IF Reporter = 0 THEN
	RETURN;
END_IF

IF _ReporterCount >= TestHarnessParameter.ReporterCapacity THEN
	THIS^.RaiseFrameworkError('the run cannot hold another reporter');
	RETURN;
END_IF

_Reporters[TO_DINT(_ReporterCount)] := Reporter;
_ReporterCount := _ReporterCount + 1;

_Fanout.Attach(Reporter);

// Suites added before this reporter was.
FOR i := 0 TO TO_DINT(_Count) - 1 DO
	THIS^.PushReporter(_Suites[i], Reporter);
END_FOR

AddReporter := TRUE;
END_METHOD

PROPERTY ReporterCount : UDINT
GET
ReporterCount := _Fanout.Count;
END_GET
END_PROPERTY

METHOD SetLabel
VAR_INPUT
	Label : T_MaxString;
END_VAR
_Label := Label;
_Tally.SetLabel(Label);
END_METHOD

// Drive the run. One suite at a time, in the order they were added.
//
// Returns TRUE once every suite has reached a terminal state.
METHOD Run : BOOL
VAR_INPUT
	Enable : BOOL;
END_VAR

VAR
	Index : DINT;
END_VAR
_Fanout.CyclicLogic();

Run := _Tally.IsComplete;

IF NOT Enable THEN
	RETURN;
END_IF

IF _IsOpen THEN
	_IsOpen := FALSE;
	THIS^.BeginTally();

	IF _Label = '' THEN
		THIS^.RaiseFrameworkError('the run was started with no label');
	END_IF

	// Once, before anything else in the run. A sink that builds something opens it
	// here rather than guessing from the first result to arrive.
	_Fanout.RunStarted(Label := _Label, TargetInfo := _TargetInfo);
END_IF

IF _Tally.IsComplete THEN
	RETURN;
END_IF

IF _Index >= TO_DINT(_Count) THEN
	THIS^.Finish();
	Run := _Tally.IsComplete;
	RETURN;
END_IF

Index := _Index;

// Serial by construction. Only one suite is ever enabled, which is what makes two
// suites touching the same axis unable to overlap.
IF _Suites[Index].Run(Enable := TRUE) THEN
	// Counts TESTS, not suites, so the figures mean the same thing at every level
	// of a nest.
	_Tally.Absorb(_Suites[Index]);
	THIS^.NextSuite();
ELSE
	THIS^.CheckWatchdog(Index);
END_IF

Run := _Tally.IsComplete;
END_METHOD

// Nothing to run. The run reports complete rather than waiting, so anything
// aggregating it is not held open.
METHOD Skip
IF NOT _IsOpen THEN
	RETURN;
END_IF

_IsOpen := FALSE;
_Tally.Begin(0);
_Index	:= TO_DINT(_Count);
THIS^.Finish();
END_METHOD

// Add a suite to the run. Order of addition is order of execution.
//
// That ordering is what gives coarse exclusion for free: two integration suites
// touching the same axis cannot overlap, because only one is ever enabled.
METHOD AddSuite : BOOL
VAR_INPUT
	Suite : I_TestSuite;
END_VAR

VAR
	Index : DINT;
	i	  : DINT;
END_VAR
AddSuite := FALSE;

IF Suite = 0 THEN
	THIS^.RaiseFrameworkError('a null suite was offered');
	RETURN;
END_IF

IF NOT _IsOpen THEN
	THIS^.RaiseFrameworkError('suites cannot be added once the run has started');
	RETURN;
END_IF

IF _Count >= Capacity THEN
	THIS^.RaiseFrameworkError('the run is full - raise its capacity argument');
	RETURN;
END_IF

Index		 := TO_DINT(_Count);
_Suites[Index] := Suite;
_Count		 := _Count + 1;

// Reporters already attached reach this suite too, so the composition root
// attaches once - to the run - whatever order it does things in.
FOR i := 0 TO TO_DINT(_ReporterCount) - 1 DO
	THIS^.PushReporter(Suite, _Reporters[i]);
END_FOR

AddSuite := TRUE;
END_METHOD

// Suites added. Assert it in CI: a suite that silently stops being added takes
// its tests with it, and the totals simply come out smaller.
PROPERTY SuiteCount : UDINT
GET
SuiteCount := _Count;
END_GET
END_PROPERTY

PROPERTY ErrorCount : UDINT
GET
ErrorCount := _Tally.ErrorCount;
END_GET
END_PROPERTY

PROPERTY FailedCount : UDINT
GET
FailedCount := _Tally.FailedCount;
END_GET
END_PROPERTY

PROPERTY IsComplete : BOOL
GET
IsComplete := _Tally.IsComplete;
END_GET
END_PROPERTY

PROPERTY Outcome : E_RunOutcome
GET
Outcome := _Tally.Outcome;
END_GET
END_PROPERTY

PROPERTY PassedCount : UDINT
GET
PassedCount := _Tally.PassedCount;
END_GET
END_PROPERTY

PROPERTY SkippedCount : UDINT
GET
SkippedCount := _Tally.SkippedCount;
END_GET
END_PROPERTY

PROPERTY TestCount : UDINT
GET
TestCount := _Tally.TestCount;
END_GET
END_PROPERTY

PROPERTY TotalDuration : LREAL
GET
TotalDuration := _Tally.TotalDuration;
END_GET
END_PROPERTY

// Start the aggregate, and re-apply anything raised before it existed.
//
// A framework error raised while the run was still OPEN - a refused suite, a
// refused reporter - has no tally to record itself into. It is counted in
// _PendingErrors and re-applied here, or a run that could not be composed
// properly reports green with its missing tests simply absent from the totals.
//
// ORDER MATTERS: Begin clears ErrorCount, so the drain must follow it. Both entry
// points into a run go through this method for that reason.
//
// _PendingErrors is NOT cleared. A suite that failed to be added is still missing
// on a re-run, so the error is re-applied every time the aggregate restarts.
METHOD BeginTally
VAR
	i : DINT;
END_VAR
_Tally.Begin(0);

FOR i := 1 TO TO_DINT(_PendingErrors) DO
	_Tally.RecordFrameworkError();
END_FOR
END_METHOD

// Has the active suite stopped making progress?
//
// PROGRESS, not duration. The measure is how many tests the suite has brought to
// a verdict - passed, failed, errored or skipped. A slow suite still moves that
// number; a stalled one does not, and counting scans since it STARTED would fire
// on the slow rather than the stuck.
//
// A suite cannot see this about itself: it is the thing that has stopped. The run
// owns the sequence, so it is the only object positioned to notice.
METHOD CheckWatchdog
VAR_INPUT
	Index : DINT;
END_VAR

VAR
	Progress : UDINT;
	Suite	 : I_TestSuite;
END_VAR
IF _WatchdogCycles = 0 THEN
	RETURN;
END_IF

Suite := _Suites[Index];

IF Suite = 0 THEN
	RETURN;
END_IF

// Every verdict the suite has reached so far.
Progress := Suite.PassedCount + Suite.FailedCount
		  + Suite.ErrorCount + Suite.SkippedCount;

IF Progress <> _LastProgress THEN
	_LastProgress := Progress;
	_StallCycles  := 0;
	RETURN;
END_IF

_StallCycles := _StallCycles + 1;

IF _StallCycles < _WatchdogCycles THEN
	RETURN;
END_IF

// Stalled. Named, counted, and left behind.
_StalledSuites := _StalledSuites + 1;
THIS^.RaiseFrameworkError(CONCAT(CONCAT(
	'suite stalled and was abandoned: ', Suite.Label),
	CONCAT(', no verdict for ', UDINT_TO_STRING(_WatchdogCycles))));

// One call with Enable FALSE, so the suite can put its own state back. Its return
// is ignored: a suite that has stopped will not answer this either, and waiting
// for it would reproduce the stall the watchdog exists to break.
Suite.Run(Enable := FALSE);

// Whatever it did manage still counts.
_Tally.Absorb(Suite);

THIS^.NextSuite();
END_METHOD

// Terminal. Settles the aggregate and raises RunFinished - ONCE, whatever the
// topology.
//
// THIS IS WHY THIS OBJECT EXISTS. A suite cannot raise it: a suite is not a run,
// and asking one to announce the end of something above itself is what forced a
// "am I being sequenced" flag in an earlier design. Here a single suite is
// composed with one TestRun and a sequencer IS one, so exactly one object is ever
// in a position to say the run is over.
METHOD Finish
IF _Tally.IsComplete THEN
	RETURN;
END_IF

_Tally.Finish();
_Fanout.RunFinished(Status := THIS^, TargetInfo := _TargetInfo);
END_METHOD

// Move to the next suite and reset the watchdog with it. One place, so the reset
// cannot be forgotten on one of the paths that advances.
METHOD NextSuite
_Index		  := _Index + 1;
_StallCycles  := 0;
_LastProgress := 0;
END_METHOD

// Hand a reporter to a suite through its configuration face.
//
// A suite is held as I_TestSuite - the driving surface - which deliberately does
// not carry AddReporter. The configuration face is reached with __QUERYINTERFACE,
// the same way every optional face in this library is.
METHOD PushReporter
VAR_INPUT
	Suite	 : I_TestSuite;
	Reporter : I_TestReporter;
END_VAR

VAR
	ConfigFace : I_TestConfiguration;
END_VAR
IF Suite = 0 THEN
	RETURN;
END_IF

IF __QUERYINTERFACE(Suite, ConfigFace) THEN
	ConfigFace.AddReporter(Reporter);
END_IF
END_METHOD

// One place run-level framework errors are named.
METHOD RaiseFrameworkError
VAR_INPUT
	Message : T_MaxString;
END_VAR
IF _IsOpen THEN
	// Before the tally exists. Held, and re-applied by BeginTally when the run
	// starts - without that, a run that could not be composed properly reports
	// green with its missing tests simply absent from the totals.
	_PendingErrors := _PendingErrors + 1;
ELSE
	_Tally.RecordFrameworkError();
END_IF

_Fanout.FrameworkError(Source := _Label, Message := Message);
END_METHOD

// Re-execute every suite in the run, and produce a FRESH document.
//
// It lives here rather than on a suite because the document boundary does. A suite
// re-running on its own re-executes its tests and raises SuiteFinished again, but
// announces no run - so no new artifact is written and the re-run is invisible to
// CI.
//
// The registered set is not redefined, at either level. A re-run re-executes what
// was composed; it does not recompose it.
//
// There is no ReRunSingle here. Re-running ONE thing is a debugging aid scoped to
// a test, and the suite already offers it - a run-level equivalent would be a
// second way to spell the same intention.
METHOD ReRun
VAR
	i		: DINT;
	ReRunFace : I_TestReRun;
END_VAR
IF _IsOpen THEN
	// Never started. There is nothing to repeat.
	RETURN;
END_IF

IF NOT _Tally.IsComplete THEN
	// Mid-run. Restarting now would leave suites half-executed and the counts
	// meaningless.
	THIS^.RaiseFrameworkError('ReRun was called while the run was still going');
	RETURN;
END_IF

FOR i := 0 TO TO_DINT(_Count) - 1 DO
	IF __QUERYINTERFACE(_Suites[i], ReRunFace) THEN
		ReRunFace.ReRun();
	END_IF
END_FOR

// Counts start again from nothing, and Finish will raise RunFinished a second
// time - which is what produces the fresh document. Anything refused at
// composition is re-applied: a suite that never made it in is still missing.
THIS^.BeginTally();
_Index		  := 0;
_StallCycles  := 0;
_LastProgress := 0;
END_METHOD

// Where this run happened - NetId, platform, TwinCAT version, whatever
// identifies the machine.
//
// Without it a matrix run across several targets produces result documents that
// cannot be told apart.
METHOD SetTargetInfo
VAR_INPUT
	TargetInfo : T_MaxString;
END_VAR
_TargetInfo := TargetInfo;
END_METHOD

// How many scans a suite may go WITHOUT COMPLETING A TEST before the run
// abandons it. Zero disables the watchdog.
//
// A backstop, not a deadline. Per-test budgets already bound every test that did
// not disable them; this catches what they cannot - a suite that stops progressing
// for any other reason, including a test that turned its own deadlines off.
//
// Raise it for a suite with a single legitimately long test: the count is scans
// between VERDICTS, so one test taking longer than the budget looks identical to
// a suite that has stopped.
METHOD SetWatchdog
VAR_INPUT
	Cycles : UDINT;
END_VAR
_WatchdogCycles := Cycles;
END_METHOD

// Suites the watchdog abandoned. Assert it is zero in CI: a stalled suite is never
// a normal outcome, and the run it belongs to cannot be trusted.
PROPERTY StalledSuites : UDINT
GET
StalledSuites := _StalledSuites;
END_GET
END_PROPERTY

END_FUNCTION_BLOCK

// Project Information/F_GetCompany
// This function has been automatically generated from the project information.
{attribute 'signature_flag' := '1073741824'}
{attribute 'TcGenerated'}
{attribute 'no-analysis'}
FUNCTION F_GetCompany : WSTRING
VAR_INPUT
	
END_VAR

F_GetCompany := "None";

END_FUNCTION

// Project Information/F_GetTitle
// This function has been automatically generated from the project information.
{attribute 'signature_flag' := '1073741824'}
{attribute 'TcGenerated'}
{attribute 'no-analysis'}
FUNCTION F_GetTitle : WSTRING
VAR_INPUT
	
END_VAR

F_GetTitle := "TestHarnessCore";

END_FUNCTION

// Project Information/F_GetVersion
// This function has been automatically generated from the project information.
{attribute 'signature_flag' := '1073741824'}
{attribute 'TcGenerated'}
{attribute 'no-analysis'}
FUNCTION F_GetVersion : ST_LibVersion
VAR_INPUT
	
END_VAR

F_GetVersion.iMajor := 0;
F_GetVersion.iMinor := 0;
F_GetVersion.iBuild := 11;
F_GetVersion.iRevision := 0;
F_GetVersion.sVersion := '0.0.11';
F_GetVersion.nFlags := 0;

END_FUNCTION
